PROGRAM LED
VAR
	
	LED1 AT%Q*: BOOL;
	SWITCH1 AT%I*: BOOL;
END_VAR

IF SWITCH1=1 THEN
	LED1:=1;
ELSE
	LED1:=0;
END_IF

END_PROGRAM

(* stored: Version 1.1.0.1, ProductVersion 3.1.4022.16
   POU LED: Id {9bc604c0-6951-44a7-a871-5e08c40d8366}, SpecialFunc None *)
